Fanuc KAREL source: kt00376.KL

PROGRAM KT00376
%STACKSIZE=65535
%PRIORITY=65535
%NOLOCKGROUP
VAR
R2 : REAL
OUT : BOOLEAN
-- UNRESOLVED DECLARATIONS (source type spelling not recovered)
-- Y1 : ARRAY[2] OF TYPE_0x0018 (type_u16=0x2018)
BEGIN
Y1[1]=2
R2=3.0
-- UNRESOLVED_PC line 10 opcodes [22 9D 33 B1 21 29 64 29 70 23] marker_code=35
END KT00376
